PROGRAM Axis01_Status
VAR
//System_Bit
	Always_ON	:	BOOL	:=TRUE	;//상시 ON 
	Always_OFF	:	BOOL	:=FALSE	;//상시 OFF
	Axis01_Status_01: MC_ReadStatus;
	Axis01_Position_Read_01: MC_ReadActualPosition;
	Axis01_Velocity_Read_01: MC_ReadActualVelocity;
	Axis01_Reset_01: MC_Reset;
	Axis01_Stop_01: MC_Stop;
END_VAR

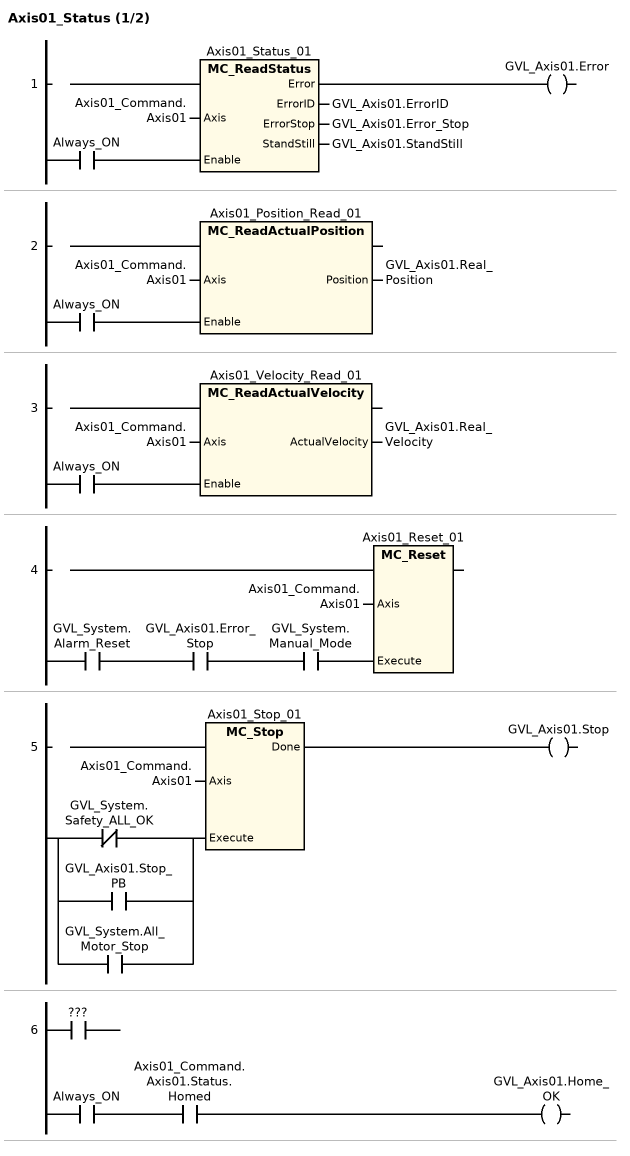
// NETWORK 1
Axis01_Status_01(
    Axis := Axis01_Command.Axis01,
    Enable := Always_ON,
    Error => GVL_Axis01.Error,
    ErrorID => GVL_Axis01.ErrorID,
    ErrorStop => GVL_Axis01.Error_Stop,
    StandStill => GVL_Axis01.StandStill); // MC_ReadStatus

// NETWORK 2
Axis01_Position_Read_01(
    Axis := Axis01_Command.Axis01,
    Enable := Always_ON,
    Position => GVL_Axis01.Real_Position); // MC_ReadActualPosition

// NETWORK 3
Axis01_Velocity_Read_01(
    Axis := Axis01_Command.Axis01,
    Enable := Always_ON,
    ActualVelocity => GVL_Axis01.Real_Velocity); // MC_ReadActualVelocity

// NETWORK 4
Axis01_Reset_01(Axis := Axis01_Command.Axis01, Execute := GVL_System.Alarm_Reset AND GVL_Axis01.Error_Stop AND GVL_System.Manual_Mode); // MC_Reset

// NETWORK 5
Axis01_Stop_01(Axis := Axis01_Command.Axis01, Execute := NOT GVL_System.Safety_ALL_OK OR GVL_Axis01.Stop_PB OR GVL_System.All_Motor_Stop); // MC_Stop
GVL_Axis01.Stop := Axis01_Stop_01.Done;

// NETWORK 6
GVL_Axis01.Home_OK := Always_ON AND Axis01_Command.Axis01.Status.Homed;

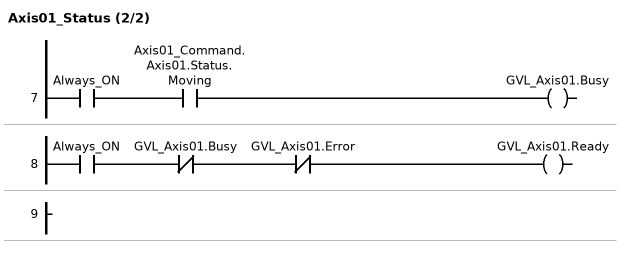
// NETWORK 7
GVL_Axis01.Busy := Always_ON AND Axis01_Command.Axis01.Status.Moving;

// NETWORK 8
GVL_Axis01.Ready := Always_ON AND NOT GVL_Axis01.Busy AND NOT GVL_Axis01.Error;

// NETWORK 9

END_PROGRAM

(* stored: Version 1.1.0.1, ProductVersion 3.1.4024.16
   POU Axis01_Status: Id {cfc680cf-dda7-423e-9182-aaaf7d5606b2}, SpecialFunc None *)
